// TIA Portal V19 export
ORGANIZATION_BLOCK "Main"   // OB3201, LAD, ProgramCycle
TITLE = "Main Program Sweep (Cycle)"
// stored: AutoNumber false, IsIECCheckEnabled true, Namespace Unit3.EM1, SetENOAutomatically true
   VAR_INPUT
      Initial_Call : Bool;   // Initial call of this OB
      Remanence : Bool;   // =True, if remanent data are available
   END_VAR
BEGIN

REGION Network 1 (SCL): mapping input

   "Unit3.EM1.instSimulation"();
END_REGION

REGION Network 2 (SCL): Call Equipment
   "Unit3.EM1.CallEquipment_DB"(unitStatus:="Unit3.EmNodes".unitStatus,
                    unitAlarmDB:="Unit3.Alarms".emAlarms[Unit3_EM1],
                    emFeedback:="Unit3.EmNodes".emFeedback[Unit3_EM1]);
END_REGION
END_ORGANIZATION_BLOCK
